(* IEC 61131-3 sources: jiepp/iec_61131-3/samples, 27 files *)

(* ---- _alarm_codes.iec ---- *)
(* _alarm_codes.iec - Alarm code fragment guarded by a classic macro guard *)
{#ifndef ALARM_CODES_INCLUDED}
{#define ALARM_CODES_INCLUDED 1}

type AlarmCode : int (
    door_open := 16#0101,
    over_pressure := 16#0102
);
end_type
{#endif}

(* ---- _io_map.iec ---- *)
(* _io_map.iec - I/O map fragment guarded by {#pragma once} *)
{#pragma once}

type IoMapInfo :
struct
    file: string := __FILE_NAME__;
    level: int := __INCLUDE_LEVEL__;
    input_count: int := 16;
end_struct;
end_type

(* ---- logging_macro.iec ---- *)
(* logging_macro.iec - Variadic logging macros using __VA_ARGS__ + @ stringize *)

{#define LOG_PREFIX(level) @level}
{#define LOG_INFO(...) log_message(LOG_PREFIX(INFO), __VA_ARGS__)}
{#define LOG_WARN(...) log_message(LOG_PREFIX(WARN), __VA_ARGS__)}
{#define LOG_ERROR(...) log_message(LOG_PREFIX(ERROR), __VA_ARGS__)}
{#define STR(x) @x}

function_block Logger
var_input
    enable: bool;
end_var
var
    msg: string[255];
end_var
if enable then
    LOG_INFO('System started');
    LOG_WARN('Low memory', ' threshold=', STR(1024));
    LOG_ERROR('Sensor failure');
end_if;
end_function_block

(* ---- nosplit.iec ---- *)
(* nosplit.iec - Forward statements that contain commas with __nosplit *)

(* GUARD takes exactly two arguments *)
{#define GUARD(cond, body) if cond then body end_if;}

(* WHEN_RUNNING forwards a whole statement block as the second argument of *)
(* GUARD. Without __nosplit, the commas in "1, 2:" would split the block    *)
(* into more arguments than GUARD takes (PP34).                            *)
{#define WHEN_RUNNING(...) GUARD(running, __nosplit(__VA_ARGS__))}

function_block Sorter
var_input
    running: bool;
    item_type: int;
end_var
var
    gate, rejected: int;
end_var
(* A call that spans several lines is output as one line; the blank lines  *)
(* after it keep the line numbers of the following code unchanged.         *)
WHEN_RUNNING(
case item_type of
1, 2: gate := 1;
3: gate := 2;
else
gate := 0; rejected := rejected + 1;
end_case;
)
end_function_block

(* ---- trace_macro.iec ---- *)
(* trace_macro.iec - Optional arguments with __VA_OPT__ and named variadic parameters *)

{#define TRACE(msg, ...) trace(__FILE_NAME__, __LINE__, msg __VA_OPT__(, __VA_ARGS__))}
{#define ALARM(code, args...) raise_alarm(code __VA_OPT__(, args))}

function_block Station
var_input
    start: bool;
end_var
var
    pressure: real;
end_var
TRACE('cycle start');
TRACE('pressure', pressure);
if not start then
    ALARM(16#0101);
    ALARM(16#0102, 'door open', pressure);
end_if;
end_function_block

(* ---- type_limits.iec ---- *)
(* type_limits.iec - Portable types and limits with built-in type macros *)

{#define COUNT_T __INT32_TYPE}
{#define FLAGS_T __BITS16_TYPE}
{#if __DINT_MAX__ > 16#7fff && defined(_JIEPP)}
{#define WIDE_COUNTER 1}
{#endif}

function_block Totalizer
var
    count: COUNT_T;
    flags: FLAGS_T;
{#ifdef WIDE_COUNTER}
    wide_total: lint;
{#endif}
end_var
if count < __DINT_MAX__ then count := count + 1; end_if;
flags := flags and __WORD_MASK__;
{#ifdef WIDE_COUNTER}
wide_total := wide_total + 1;
{#endif}
end_function_block

(* ---- xml_output.iec ---- *)
(* xml_output.iec - Write LD XML through macros with __xmlattr, __xmltext and __arg_* *)

(* CONTACT puts its operand into an XML attribute. __xmlattr quotes the text *)
(* and escapes & < > " ' so that the attribute stays well-formed XML.        *)
{#define CONTACT(op) <LdObject xsi:type="Contact" operand=__xmlattr(op)/>}

(* NOTE puts its text into element content. __xmltext escapes & < > only. *)
{#define NOTE(t) <Comment>__xmltext(t)</Comment>}

(* ARG splits a call argument "pin := value" (input) or "pin => var" (output) *)
(* at the first separator. __arg_lhs is the pin, __arg_rhs is the value or    *)
(* the variable, and __arg_dir is 0 for ":=" and 1 for "=>". The __xmlattr    *)
(* around each part quotes it, including the number from __arg_dir.           *)
{#define ARG(a) <Arg name=__xmlattr(__arg_lhs(a)) dir=__xmlattr(__arg_dir(a)) value=__xmlattr(__arg_rhs(a))/>}

(* CALL_TON is an FB call. The two arguments become two <Arg> elements. *)
{#define CALL_TON(inst, pt, q) <Block xsi:type="FbCall" instance=__xmlattr(inst)>ARG(pt) ARG(q)</Block>}

function_block Timer
var_input
    start: bool;
    mode: string;
end_var
var_output
    done: bool;
end_var
var
    delay: time;
    ton1: ton;
end_var
{ld}
CONTACT(mode = 'RUN' & start)
CONTACT(delay < T#10s)
CALL_TON(ton1, PT := T#2s, Q => done)
NOTE(done is set when delay < 2s & start = true)
{end}
end_function_block

(* ---- assert.iec ---- *)
(* assert.iec - Expansion-time checks with __assert, __error and __has_builtin *)

{#define AXIS_COUNT 4}
{#define MAX_AXES 8}
{#define CYCLE_TIME_MS 10}

(* A check outside any macro expands to nothing when it holds *)
__assert(AXIS_COUNT <= MAX_AXES, too many axes: AXIS_COUNT > MAX_AXES)
__assert(defined(CYCLE_TIME_MS), CYCLE_TIME_MS must be defined)

(* Directives cannot be written in a macro body, but __assert can. The   *)
(* check runs at each use; parameter names in the message are replaced, *)
(* so AXIS_TABLE(axes, 12) reports 'axes has 12 entries, allowed 1 to 8' *)
{#define AXIS_TABLE(name, size) __assert(size >= 1 && size <= MAX_AXES, name has size entries, allowed 1 to MAX_AXES)name: array[1..size] of AxisRef}

(* -D '__assert(...)=' turns the checks off; __has_builtin tells whether they run *)
{#if __has_builtin(__assert)}
{#define CHECKS_ACTIVE true}
{#else}
{#define CHECKS_ACTIVE false}
{#endif}

(* __error reports only when the macro that contains it is used *)
{#if defined(TARGET_OMRON) || defined(TARGET_SIEMENS)}
{#define HIGH_SPEED_COUNTER(name) name: HscCounter}
{#else}
{#define HIGH_SPEED_COUNTER(name) __error(HIGH_SPEED_COUNTER is not supported on this target)}
{#endif}

program Main
var
    AXIS_TABLE(axes, AXIS_COUNT);
    checks_active: bool := CHECKS_ACTIVE;
    cycle_ms: int := CYCLE_TIME_MS;
end_var
end_program

(* ---- builtin_macros.iec ---- *)
(* builtin_macros.iec - Built-in macros *)

program Main
var
    line_num: int;
    inc_level: int;
    counter1, counter2, counter3: int;
    file_name: string[255];
    file_name_only: string[255];
    base_name: string[255];
end_var
line_num := __LINE__;
inc_level := __INCLUDE_LEVEL__;
file_name := __FILE__;
file_name_only := __FILE_NAME__;
base_name := __BASE_FILE__;
counter1 := __COUNTER__;
counter2 := __COUNTER__;
counter3 := __COUNTER__;
{#if __has_include('_header.iec')}
(* _header.iec exists *)
{#include '_header.iec'}
{#endif}
end_program

(* ---- conditional.iec ---- *)
(* conditional.iec - Conditional compilation *)

{#define TARGET_OMRON 1}

{#ifdef TARGET_OMRON}
{#define TIMER_FB TON}
{#else}
{#define TIMER_FB Timer}
{#endif}

{#ifndef DEBUG}
{#define DEBUG 0}
{#endif}

{#if defined(TARGET_OMRON) && DEBUG = 1}
{#define LOG_ENABLED 1}
{#elif defined(TARGET_OMRON)}
{#define LOG_ENABLED 0}
{#else}
{#define LOG_ENABLED 0}
{#endif}

program Main
var
    t1: TIMER_FB;
    log_flag: int;
end_var
log_flag := LOG_ENABLED;
end_program

(* ---- define.iec ---- *)
(* define.iec - Object macros and #undef *)

{#define PI 3.14159}
{#define GRAVITY 9.81}

program Main
var
    r, area, force, mass: lreal;
end_var
area := PI * r * r;
{#undef PI}
{#define PI 3.14}
area := PI * r * r;
force := mass * GRAVITY;
end_program

(* ---- error_warning.iec ---- *)
(* error_warning.iec - #error, #warning and #info *)

{#define PLATFORM_DEFINED 1}

{#ifndef PLATFORM_DEFINED}
{#error 'PLATFORM_DEFINED is not set'}
{#endif}

{#if 0}
(* This block is not evaluated, so #error will not occur *)
{#error 'This should never trigger'}
{#endif}

{#warning 'This is a compile-time warning'}

{#info 'This is an informational message'}

program Main
end_program

(* ---- function_macro.iec ---- *)
(* function_macro.iec - Function macros *)

{#define MAX2(a, b) SEL((a) > (b), (b), (a))}
{#define CLAMP(v, lo, hi) MAX2(lo, SEL((v) > (hi), (v), (hi)))}

program Main
var
    x, y, result: int;
end_var
result := MAX2(x, y);
result := CLAMP(x, 0, 100);
end_program

(* ---- generic_function.iec ---- *)
(* generic_function.iec - Generate type-parameterized functions using @@ and function macros *)

{#define DECL_ADD(T)
function add_@@T: T$n$
var_input$n$
	in1, in2: T;$n$
end_var$n$
add_@@T := in1 + in2;$n$
end_function
}

DECL_ADD(int);
DECL_ADD(dint);
DECL_ADD(lreal);

program Main
var
	i: int;
	d: dint;
	r: lreal;
end_var
i := add_int(1, 2);
d := add_dint(100, 200);
r := add_lreal(1.5, 2.5);
end_program

(* ---- ignore.iec ---- *)
(* ignore.iec - Suppress error codes with #ignore *)

(* Suppress the PP49 warning (extra tokens after {#endif}) for the *)
(* legacy-style labelled {#endif TARGET_X} below *)
{#ignore PP49}

{#ifdef TARGET_X}
{#define LEGACY_FLAG 1}
{#endif TARGET_X}

program Main
end_program

(* ---- include.iec ---- *)
(* include.iec — #include: relative path ('...') and system path (<...>) *)

(* 'file' form: searches relative to current file, then system paths *)
(* Same as GCC #include "file" *)
{#include '_header.iec'}

(* <file> form: searches system paths only *)
(* Same as GCC #include <file> — equivalent to {#sinclude 'file'} *)
{#syspath 'lib'}
{#include <_util.iec>}

program Main
var
    buf: string[MAX_BUFFER_SIZE];
    ver: int;
    loaded: int;
end_var
ver := VERSION;
loaded := UTIL_LOADED;
end_program

(* ---- include_guard.iec ---- *)
(* include_guard.iec - Include guards: {#pragma once} and macro guard *)

(* Each fragment is included twice. {#pragma once} skips the whole file on  *)
(* the second include. A macro guard skips only the text between {#ifndef}  *)
(* and {#endif}; the header comment before the guard is emitted again.      *)
{#include '_io_map.iec'}
{#include '_io_map.iec'}
{#include '_alarm_codes.iec'}
{#include '_alarm_codes.iec'}

program Main
var
    info: IoMapInfo;
    alarm: AlarmCode := AlarmCode#door_open;
end_var
end_program

(* ---- macro_rescan.iec ---- *)
(* macro_rescan.iec - arguments are rescanned, __VA_OPT__ looks at the expanded argument *)

{#define EMPTY}
{#define LPAREN (}
{#define DEFER(id) id EMPTY}
{#define EXPAND(...) __VA_ARGS__}
{#define TWICE(x) (x) * 2}

(* __VA_OPT__ keeps its content only when the expanded variable arguments are not empty. *)
{#define LOG(fmt, ...) log(fmt __VA_OPT__(,) __VA_ARGS__)}

program Main
var
    n: int;
end_var
(* DEFER hides the call from the first scan; EXPAND scans it again. *)
n := DEFER(TWICE)(3);
n := EXPAND(DEFER(TWICE)(3));
LOG('start');
LOG('empty', EMPTY);
LOG('value', n);
end_program

(* ---- named_counter.iec ---- *)
(* named_counter.iec - Independent numbering with __counter, __counter_peek and __counter_set *)

(* Each DETECT gets the next slot of edge_trig[]. The slot number is passed  *)
(* through a parameter, so both uses in DETECT_ see the same value.          *)
{#define EDGE_SLOTS 8}
{#define DETECT_(sig, q, i) edge_trig[i](CLK := sig); q := edge_trig[i].Q}
{#define DETECT(sig, q) DETECT_(sig, q, __counter(edge))}

(* Alarm numbers start at 100 and do not share numbers with the edge slots *)
__counter_set(alarm, 100)
{#define NEXT_ALARM() __counter(alarm)}

program Main
var
    start_button, stop_button, door_switch: bool;
    start_pressed, stop_pressed, door_opened: bool;
    edge_trig: array[0..EDGE_SLOTS - 1] of R_TRIG;
    door_alarm, overload_alarm: int;
    used_slots: int;
end_var
DETECT(start_button, start_pressed);
DETECT(stop_button, stop_pressed);
DETECT(door_switch, door_opened);
door_alarm := NEXT_ALARM();
overload_alarm := NEXT_ALARM();
(* __counter_peek reads a counter without advancing it *)
used_slots := __counter_peek(edge);
__assert(__counter_peek(edge) <= EDGE_SLOTS, more DETECT uses than EDGE_SLOTS)
end_program

(* ---- platform_switch.iec ---- *)
(* platform_switch.iec - Multi-platform switching with #if/#elif *)

{#define TARGET_OMRON 1}

{#if defined(TARGET_OMRON)}
  {#define FB_TIMER TON}
  {#define FB_COUNTER CTU}
  {#define MAX_IO 2048}
{#elif defined(TARGET_MITSUBISHI)}
  {#define FB_TIMER Timer_100ms}
  {#define FB_COUNTER UpCounter}
  {#define MAX_IO 1024}
{#elif defined(TARGET_SIEMENS)}
  {#define FB_TIMER TON_TIME}
  {#define FB_COUNTER CTU_INT}
  {#define MAX_IO 4096}
{#else}
  {#error 'Unknown target platform. Define TARGET_OMRON, TARGET_MITSUBISHI, or TARGET_SIEMENS.'}
{#endif}

program Main
var
    timer1: FB_TIMER;
    counter1: FB_COUNTER;
    io_count: int;
end_var
io_count := MAX_IO;
end_program

(* ---- pp_number.iec ---- *)
(* pp_number.iec - a number with letters after it is one token *)

(* Macros named like the units of a time literal ... *)
{#define ms 1000}
{#define s 60}

program Main
var
    t: time;
    n: int;
end_var
(* ... do not expand inside the literal: t#10ms and t#1m30s stay as written. *)
t := t#10ms;
t := t#1m30s;
(* A separate name still expands. *)
n := ms;
n := s;
end_program

(* ---- pragma.iec ---- *)
(* pragma.iec - Runtime limit directives ({#max_*}) *)

{#max_expansion_depth 128}
{#max_if_nesting 64}
{#max_include_depth 100}

{#define X 42}

program Main
var
    v: int;
end_var
v := X;
end_program

(* ---- setline.iec ---- *)
(* setline.iec - Set line numbers with #line / #set_line *)

{#line 100}

program Main
var
    line_a, line_b: int;
end_var
line_a := __LINE__;
{#set_line 200 'virtual.iec'}
line_b := __LINE__;
end_program

(* ---- stringize.iec ---- *)
(* stringize.iec - @ stringification operator *)

{#define STR(x) @x}

program Main
var
    s1, s2, s3: string[255];
    ws: wstring;
end_var
s1 := STR(Hello World);
s2 := {## 123 + 456};
s3 := {## __LINE__};
ws := {#wstring Hello World};
end_program

(* ---- syspath.iec ---- *)
(* syspath.iec — #syspath + #sinclude: system-path-only include *)
(* #sinclude searches system paths only, equivalent to #include <...> *)

{#syspath 'lib'}
{#sinclude '_util.iec'}

program Main
var
    v: int;
end_var
v := ABS_OF(-10);
end_program

(* ---- token_paste.iec ---- *)
(* token_paste.iec - @@ token concatenation operator *)

{#define VAR_NAME(prefix, n) prefix@@_@@n}
{#define TYPED(type, suffix) type@@suffix}

(* Unique instance names: the extra level expands __COUNTER__ before pasting *)
{#define CAT_(a, b) a@@b}
{#define CAT(a, b) CAT_(a, b)}
{#define UNIQUE(p) CAT(p, __COUNTER__)}

program Main
var
    VAR_NAME(sensor, 1): int;
    VAR_NAME(sensor, 2): int;
    v: TYPED(d, int);
    UNIQUE(ton_): TON;
    UNIQUE(ton_): TON;
end_var
VAR_NAME(sensor, 1) := 100;
VAR_NAME(sensor, 2) := 200;
end_program

(* ---- variadic.iec ---- *)
(* variadic.iec - __VA_ARGS__ and __VA_ARGC__ *)

{#define PRINT(...) print(__VA_ARGS__)}
{#define COUNT(...) __VA_ARGC__}
{#define FIRST(a, ...) a}
{#define REST(a, ...) __VA_ARGS__}

program Main
var
    n: int;
end_var
PRINT(1, 2, 3);
n := COUNT(a, b, c);
n := FIRST(10, 20, 30);
PRINT(REST(1, 2, 3));
end_program
